(* IEC 61131-3 sources: programs/VI-54/VI-54_20171205/VI-54_20171205/Stations/Screen/LseClass170718/Class/Comm_SendData, 1 file *)

(* ---- Comm_SendData.st ---- *)
(*!
<Class
	Name               = "Comm_SendData"
	Revision           = "0.5"
	RealtimeTask       = "false"
	CyclicTask         = "false"
	BackgroundTask     = "false"
	Sigmatek           = "false"
	OSInterface        = "false"
	HighPriority       = "false"
	Automatic          = "false"
	UpdateMode         = "Prescan"
	SharedCommandTable = "true"
	Objectsize         = "(600,360)"
	Comment            = "Sending data via communication class.">
	<Channels>
		<Server Name="ClassSvr" Visualized="false" Initialize="false" WriteProtected="false" Retentive="false"/>
		<Server Name="sDestinationId" Visualized="false" Initialize="true" WriteProtected="true" Retentive="false" Comment="Destination communication id number."/>
		<Server Name="sMyId" Visualized="false" Initialize="true" WriteProtected="true" Retentive="false" Comment="Source communication id number."/>
		<Server Name="sSendCnt" Visualized="false" Initialize="false" WriteProtected="false" Retentive="false" Comment="Counter for sended data blocks."/>
		<Server Name="sSendErr" Visualized="false" Initialize="false" WriteProtected="false" Retentive="false" Comment="Counter for send errors."/>
		<Client Name="cDataMng" Required="true" Internal="false" Comment="Connection to communication data manager."/>
		<Client Name="cPrio" Required="true" Internal="false" Comment="Communication priority number."/>
		<Client Name="cSendErr" Required="false" Internal="false" Comment="Write out JobID if sending was not Ok."/>
		<Client Name="cSendOk" Required="false" Internal="false" Comment="Write out JobID if sending was Ok."/>
	</Channels>
	<RevDoku>
		<Owner/>
		<Dokumentation Revision="0.5" Date="2014-12-03" Author="W.Brunner" Company="DETS" Description="Added GetOnlineState() method."/>
		<Dokumentation Revision="0.4" Date="2014-12-03" Author="hötant" Company="DETS" Description="added some Trace messages "/>
		<Dokumentation Revision="0.3" Date="2014-11-11" Author="hötant" Company="DETS" Description="added optional parameter to method SendData"/>
		<Dokumentation Revision="0.2" Date="2014-10-21" Author="hötant" Company="DETS" Description="added _MNG_GlobalReciveError in method CallBackJobState"/>
		<Dokumentation Revision="0.1" Date="2014-10-17" Author="W.Brunner" Company="DETS" Description="Deleted retry. Added callback error detection."/>
	</RevDoku>
</Class>
*)
Comm_SendData : CLASS
  //Servers:
	ClassSvr 	: SvrChCmd_DINT;
	sMyId 	: SvrCh_DINT;
	sDestinationId 	: SvrCh_DINT;
	sSendCnt 	: SvrCh_DINT;
	sSendErr 	: SvrCh_DINT;
  //Clients:
	cDataMng 	: CltChCmd_DataManager;
	cPrio 	: CltCh_DINT;
	cSendOk 	: CltCh_DINT;
	cSendErr 	: CltCh_DINT;
  //Variables:
  //Functions:

	FUNCTION VIRTUAL GLOBAL Init;

	FUNCTION VIRTUAL GLOBAL CallBackJobState
		VAR_INPUT
			JobID 	: DINT;
			JobState 	: DINT;
		END_VAR;

	FUNCTION VIRTUAL GLOBAL SendData
		VAR_INPUT
			pData 	: ^void;
			length 	: UDINT;
			timeout 	: UDINT;
			OptCMD 	: USINT := 0;
		END_VAR
		VAR_OUTPUT
			JobID 	: DINT;
		END_VAR;

	FUNCTION GLOBAL GetOnlineState
		VAR_OUTPUT
			retcode 	: BOOL;
		END_VAR;
  //Tables:
	FUNCTION @STD
		VAR_OUTPUT
			ret_code	: CONFSTATES;
		END_VAR;
	FUNCTION GLOBAL TAB @CT_;
END_CLASS;

#pragma usingLtd DataManager

FUNCTION GLOBAL Comm_SendData_CB
	VAR_INPUT
		pthis 	: ^void;
		JobID 	: DINT;
		JobState 	: DINT;
	END_VAR

  pthis$^Comm_SendData^.CallBackJobState(JobID, JobState);

END_FUNCTION

FUNCTION VIRTUAL GLOBAL Comm_SendData::CallBackJobState
	VAR_INPUT
		JobID 	: DINT;
		JobState 	: DINT;
	END_VAR
  var
    txt1 : array [0..199] of char;
    txt2 : array [0..199] of char;
    txtOut : array [0..599] of char;
    mError : usint;
  END_VAR

  mError :=0;
  case JobState$DataManagerPriority::t_e_CallbackState of
    //Ok
    _MNG_Received:
       cSendOk :=JobID;
       cSendOk.write (cSendOk);

    //Error
    _MNG_NoReceiverConnected:
       cSendErr :=JobId;
       cSendErr.write (cSendErr);
       sSendErr +=1;
       _strcpy(dest:=#txt1[0], src:="_MNG_NoReciverConnected");
       mError :=1;
    _MNG_GlobalReceiveError:
       cSendErr :=JobId;
       cSendErr.write (cSendErr);
       sSendErr +=1;
       _strcpy(dest:=#txt1[0], src:="_MNG_GlobalReciveError");
       mError :=1;
    _MNG_TimeOut:
       cSendErr :=JobId;
       cSendErr.write (cSendErr);
       sSendErr +=1;
       _strcpy(dest:=#txt1[0], src:="_MNG_TimeOut");
       mError :=1;

  end_case;

  if mError <> 0 then
    _GetObjName(pThis:=this, pName:=#txt2[0]);
    _strcpy(dest:=#txtout[0], src:=#txt2[0]);
    _strcat(dest:=#txtout[0], src:="-> CallBackJobState -> ");
    _strcat(dest:=#txtout[0], src:=#txt1[0]);
    TRACE(#txtout[0]);
  end_if;

END_FUNCTION

FUNCTION VIRTUAL GLOBAL Comm_SendData::Init

  if _FirstScan then
  end_if;

END_FUNCTION

FUNCTION VIRTUAL GLOBAL Comm_SendData::SendData
	VAR_INPUT
		pData 	: ^void;
		length 	: UDINT;
		timeout 	: UDINT;
		OptCMD 	: USINT;(* := 0 *)
	END_VAR
	VAR_OUTPUT
		JobID 	: DINT;
	END_VAR
  VAR
  	tmpDestinationID: DINT;
    txt1 : array [0..199] of char;
    txt2 : array [0..99] of char;
    txtOut : array [0..599] of char;
  END_VAR

  // refresh online state
    GetOnlineState();

  tmpDestinationID := to_dint(OptCMD);
  tmpDestinationID := tmpDestinationID shl 24;
  tmpDestinationID := tmpDestinationID OR ( sDestinationId AND 16#00FFFFFF );

  cPrio := cPrio.Read();
  Jobid := cDataMng.SetData(  dDestinationID:= tmpDestinationID,
                              dSourceID:=      sMyId,
                              pData:=         pData,
                              udSize:=        length,
                              pThis:=         this,
                              pCallBack:=     #Comm_SendData_CB(),
                              udTimeOut:=     timeout,
                              dPrio:=          cPrio);

  if JobID <0 then
    sSendErr +=1;
    case JobID of
      -1 :  _strcpy(dest:=#txt1[0], src:="Buffer Problem !");
      -2 :  _strcpy(dest:=#txt1[0], src:="Offline !");
      -3 :  _strcpy(dest:=#txt1[0], src:="Priorität nicht gültig !");
      -4 :  _strcpy(dest:=#txt1[0], src:="Aufruf aus RT nicht erlaubt !");
    else
      _strcpy(dest:=#txt1[0], src:="Retcode nicht bekannt !");
    end_case;
    _GetObjName(pThis:=this, pName:=#txt2[0]);
    _strcpy(dest:=#txtout[0], src:=#txt2[0]);
    _strcat(dest:=#txtout[0], src:="-> SendData -> ");
    _strcat(dest:=#txtout[0], src:=#txt1[0]);
    TRACE(#txtout[0]);
  else
    sSendCnt +=1;
  end_if;

END_FUNCTION

FUNCTION GLOBAL Comm_SendData::GetOnlineState
	VAR_OUTPUT
		retcode 	: BOOL;
	END_VAR

  retcode :=cDataMng.GetOnlineState();
  if retcode =true then
     ClassSvr :=1;
  else
     ClassSvr :=0;
  end_if;

END_FUNCTION
